TYPE ST_MCHMIPrepareScreen_01_XX :
STRUCT
	btmpValue_01_XX	: BOOL;
END_STRUCT
END_TYPE

(* stored: Version 1.1.0.1
   DUT ST_MCHMIPrepareScreen_01_XX: Id {e5c41a77-0f06-04e9-1d51-b2d6d911a624} *)
